FUNCTION F_LimitTarget : DINT //used to translate EtherCAT communication from RAW variables to Kid Variables

VAR_INPUT
	Target : DINT;
END_VAR
VAR
	CorrectedTarget : DINT;
	ho: INT;
	Resulting_Max : DINT;
	Resulting_Min : DINT;
	posi: INT;
END_VAR


CorrectedTarget := GVL_index.Home_Offset;
CorrectedTarget := KidAxis.actualPos;
CorrectedTarget := KidAxis.HomedPosition_toMom;
CorrectedTarget := Target ;

IF KidAxis.IsUltimateLimitBypassed THEN 
	F_LimitTarget := Target;
	RETURN;
END_IF

IF SetAdminMax THEN GVL_Index.Admin_Max := KidAxis.actualPos; SetAdminMax := FALSE; END_IF
IF SetAdminMin THEN GVL_Index.Admin_Min := KidAxis.actualPos; SetAdminMin := FALSE;END_IF	
IF SetUserMax AND KidAxis.HomedPosition_toMom > GVL_Index.User_Max_UU THEN GVL_Index.User_Max_UU := KidAxis.HomedPosition_toMom; SetUserMax:=FALSE; END_IF
IF SetUserMin AND KidAxis.HomedPosition_toMom > GVL_Index.User_Min_UU THEN GVL_Index.User_Min_UU := KidAxis.HomedPosition_toMom; SetUserMin:= FALSE; END_IF

IF GVL_HMI.BlowOutLimits THEN
	GVL_Index.Admin_Max := 2147483647;
	GVL_Index.Admin_Min := -2147483648;
	GVL_Index.User_Max_UU := 32000;
	GVL_Index.User_Min_UU := -32000;
	GVL_HMI.BlowOutLimits := FALSE;
END_IF

		
//ADMIN LIMITS
 
IF NOT GVL_Index.Direction_Flipped THEN
	IF GVL_Index.Home_Offset + (GVL_Index.User_Min_UU *LREAL_TO_INT(1/ GVL_Motion.lrEncoder_ScalingNum))< GVL_Index.admin_Min THEN GVL_Index.User_Min_UU := (GVL_Index.Admin_Min -GVL_Index.Home_Offset)/LREAL_TO_INT(1/ GVL_Motion.lrEncoder_ScalingNum); END_IF
	IF GVL_Index.Home_Offset + (GVL_Index.User_Max_UU *LREAL_TO_INT(1/ GVL_Motion.lrEncoder_ScalingNum))> GVL_Index.admin_Max THEN GVL_Index.User_Max_UU := (GVL_Index.Admin_Max -GVL_Index.Home_Offset)/LREAL_TO_INT(1/ GVL_Motion.lrEncoder_ScalingNum); END_IF
	Resulting_Max := GVL_Index.Home_Offset + (GVL_Index.User_Max_UU *LREAL_TO_INT(1/ GVL_Motion.lrEncoder_ScalingNum));
	Resulting_Min := GVL_Index.Home_Offset + (GVL_Index.User_Min_UU *LREAL_TO_INT(1/ GVL_Motion.lrEncoder_ScalingNum));
	IF CorrectedTarget > KidAxis.actualPos AND  (NOT GVL_Safe_IO.bLimit_Hard_Up AND NOT GVL_Safe_IO.bHard_Up_Bypass_Enable) THEN CorrectedTarget := KidAxis.actualPos; END_IF
	IF CorrectedTarget < KidAxis.actualPos AND  (NOT GVL_Safe_IO.bLimit_Hard_down AND NOT GVL_Safe_IO.bHard_DOWN_Bypass_Enable) THEN CorrectedTarget := KidAxis.actualPos; END_IF
ELSE
	IF GVL_Index.Home_Offset + (GVL_Index.User_Max_UU *LREAL_TO_INT(1/ GVL_Motion.lrEncoder_ScalingNum))< GVL_Index.admin_Min THEN GVL_Index.User_Max_UU := (GVL_Index.Admin_Min -GVL_Index.Home_Offset)/LREAL_TO_INT(1/ GVL_Motion.lrEncoder_ScalingNum); END_IF
	IF GVL_Index.Home_Offset + (GVL_Index.User_Min_UU *LREAL_TO_INT(1/ GVL_Motion.lrEncoder_ScalingNum))> GVL_Index.admin_Max THEN GVL_Index.User_Min_UU := (GVL_Index.Admin_Max -GVL_Index.Home_Offset)/LREAL_TO_INT(1/ GVL_Motion.lrEncoder_ScalingNum); END_IF
	Resulting_Min:= GVL_Index.Home_Offset + (GVL_Index.User_Max_UU *LREAL_TO_INT(1/ GVL_Motion.lrEncoder_ScalingNum));
	Resulting_Max := GVL_Index.Home_Offset + (GVL_Index.User_Min_UU *LREAL_TO_INT(1/ GVL_Motion.lrEncoder_ScalingNum));
	IF CorrectedTarget < KidAxis.actualPos AND  (NOT GVL_Safe_IO.bLimit_Hard_Up AND NOT GVL_Safe_IO.bHard_Up_Bypass_Enable) THEN CorrectedTarget := KidAxis.actualPos; END_IF
	IF CorrectedTarget > KidAxis.actualPos AND  (NOT GVL_Safe_IO.bLimit_Hard_down AND NOT GVL_Safe_IO.bHard_DOWN_Bypass_Enable) THEN CorrectedTarget := KidAxis.actualPos; END_IF
END_IF

IF NOT bLimit_Software_Bypass THEN
	IF CorrectedTarget > Resulting_Max THEN CorrectedTarget := Resulting_Max; END_IF
	IF CorrectedTarget < Resulting_Min THEN CorrectedTarget := Resulting_Min ; END_IF
END_IF

kidAxis.ActiveTarget := CorrectedTarget;
F_LimitTarget := CorrectedTarget;

RETURN ;

END_FUNCTION

(* stored: Version 1.1.0.1, ProductVersion 3.1.4022.7
   POU F_LimitTarget: Id {c0951656-a73d-4dc9-a349-86341241d53c}, SpecialFunc None *)
